TYPE DUT_SQL :
STRUCT
    SensorValue : INT;
    SampleNr : INT;
    Timestamp : STRING(50);
END_STRUCT
END_TYPE

(* stored: Version 1.1.0.1
   DUT DUT_SQL: Id {bec8ac02-1e7c-4483-9698-bf94b7e943f6} *)
